PROGRAM MAIN
VAR

END_VAR

PLC_PRG();

END_PROGRAM

(* stored: Version 1.1.0.1, ProductVersion 3.1.4022.12
   POU MAIN: Id {fa451cd0-229a-43d7-b45d-a11532858704}, SpecialFunc None *)
